SUBAPPLICATION mapping_Uebung_006c (* SR-Flip-Flop mit IB auf DI_REPEAT *)
  (* Standard: 61499-2; Description: Copyright (c) 2023 Meisterschulen am Ostbahnhof This program and the accompanying materials are made available under the terms of the Eclipse Public License 2.0 which is available at https://www.eclipse.org/legal/epl-2.0/ SPDX-License-Identifier: EPL-2.0 *)
  (* Version 1.0, 2023-10-23, Franz Höpfinger, Meisterschulen am Ostbahnhof *)
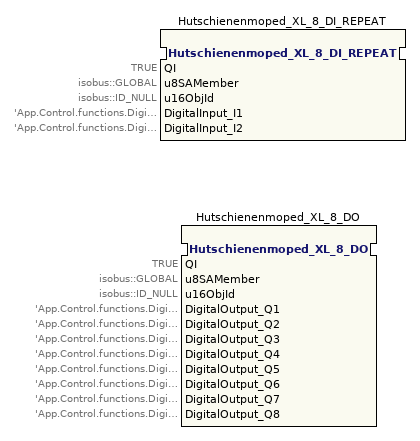
  FBS
    Hutschienenmoped_XL_8_DO : Hutschienenmoped_XL_8_DO(QI := TRUE, u8SAMember := isobus::GLOBAL, u16ObjId := isobus::ID_NULL, DigitalOutput_Q1 := 'App.Control.functions.DigitalOutput_Q1', DigitalOutput_Q2 := 'App.Control.functions.DigitalOutput_Q2', DigitalOutput_Q3 := 'App.Control.functions.DigitalOutput_Q3', DigitalOutput_Q4 := 'App.Control.functions.DigitalOutput_Q4', DigitalOutput_Q5 := 'App.Control.functions.DigitalOutput_Q5', DigitalOutput_Q6 := 'App.Control.functions.DigitalOutput_Q6', DigitalOutput_Q7 := 'App.Control.functions.DigitalOutput_Q7', DigitalOutput_Q8 := 'App.Control.functions.DigitalOutput_Q8');
    Hutschienenmoped_XL_8_DI_REPEAT : Hutschienenmoped_XL_8_DI_REPEAT(QI := TRUE, u8SAMember := isobus::GLOBAL, u16ObjId := isobus::ID_NULL, DigitalInput_I1 := 'App.Control.functions.DigitalInput_RPT_I1', DigitalInput_I2 := 'App.Control.functions.DigitalInput_RPT_I2');
  END_FBS
END_SUBAPPLICATION
